// Mitsubishi GX Works2 project: 4Pump_v1   PLC: FX3U/FX3UC

PROGRAM MAIN
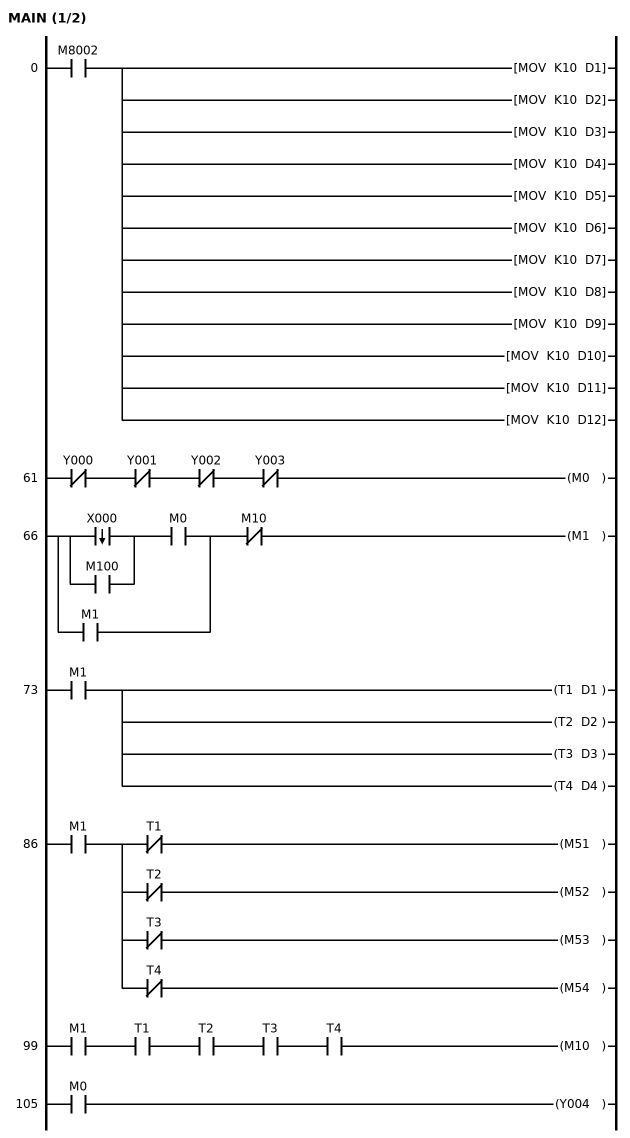
0     LD      M8002
      MOV     K10 D1
      MOV     K10 D2
      MOV     K10 D3
      MOV     K10 D4
      MOV     K10 D5
      MOV     K10 D6
      MOV     K10 D7
      MOV     K10 D8
      MOV     K10 D9
      MOV     K10 D10
      MOV     K10 D11
      MOV     K10 D12
61    LDI     Y000
      ANI     Y001
      ANI     Y002
      ANI     Y003
      OUT     M0
66    LDF     X000
      OR      M100
      AND     M0
      OR      M1
      ANI     M10
      OUT     M1
73    LD      M1
      OUT     T1 D1
      OUT     T2 D2
      OUT     T3 D3
      OUT     T4 D4
86    LD      M1
      MPS
      ANI     T1
      OUT     M51
      MRD
      ANI     T2
      OUT     M52
      MRD
      ANI     T3
      OUT     M53
      MPP
      ANI     T4
      OUT     M54
99    LD      M1
      AND     T1
      AND     T2
      AND     T3
      AND     T4
      OUT     M10
105   LD      M0
      OUT     Y004
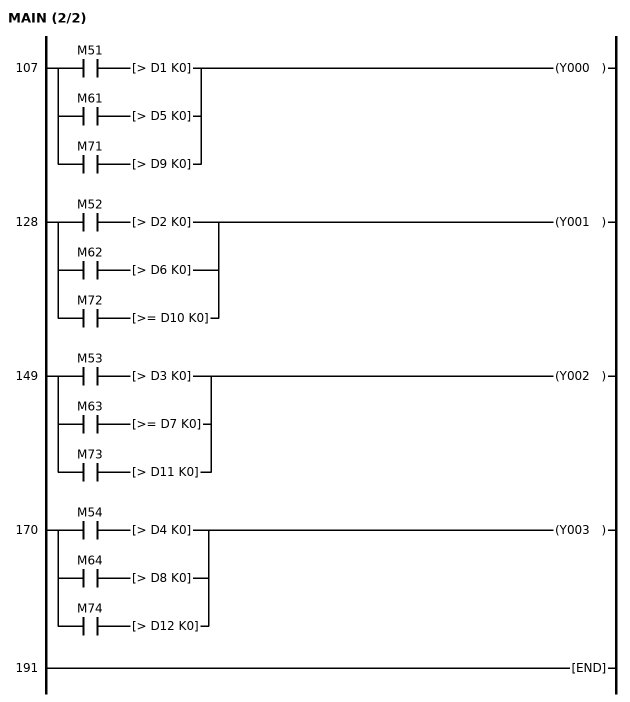
107   LD      M51
      AND>    D1 K0
      LD      M61
      AND>    D5 K0
      ORB
      LD      M71
      AND>    D9 K0
      ORB
      OUT     Y000
128   LD      M52
      AND>    D2 K0
      LD      M62
      AND>    D6 K0
      ORB
      LD      M72
      AND>=   D10 K0
      ORB
      OUT     Y001
149   LD      M53
      AND>    D3 K0
      LD      M63
      AND>=   D7 K0
      ORB
      LD      M73
      AND>    D11 K0
      ORB
      OUT     Y002
170   LD      M54
      AND>    D4 K0
      LD      M64
      AND>    D8 K0
      ORB
      LD      M74
      AND>    D12 K0
      ORB
      OUT     Y003
191   END
END_PROGRAM
